RoboDK station: Pick and Place TT.rdk

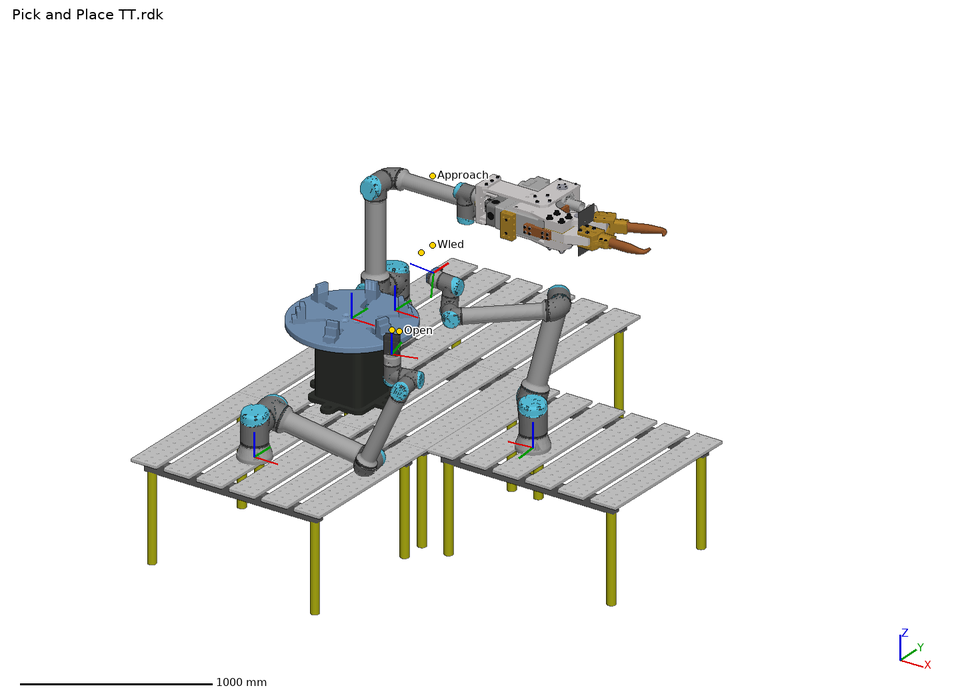
[picture v0: the station drawn from its stored meshes, robots at their saved joint values, targets as dots, program paths as lines]
Station Pick and Place (saved by RoboDK 5.6.0). Poses are relative to the parent item; angles as X-Y-Z fixed-axis rotations.
  - object Table at (1940, 2070, 0) mm, size 1193.8 x 965.2 x 609.6 mm, geometry from welding_table.sld
  - object Table at (740, 2070, 0) mm, size 1193.8 x 965.2 x 609.6 mm, geometry from welding_table.sld
  - object Table at (740, 3040, 0) mm, size 1193.8 x 965.2 x 609.6 mm, geometry from welding_table.sld
  - object Table at (740, 1100, 0) mm, size 1193.8 x 965.2 x 609.6 mm, geometry from welding_table.sld
  - frame UR10e Base at (660, 1000, 0) mm
    - robot UR10e: 6 axes, payload 10 kg, reach 1300 mm, repeatability 0.05 mm, weight 28.9 kg
        modified DH rows (alpha deg, a mm, theta deg, d mm): 0, 0, 0, 180.7; 90, 0, 180, 0; 0, 612.6, 0, 0; 0, 571.335, 0, 174.15; -90, 0, 0, 119.85; 90, 0, 180, 116.55
        joint limits [-360, -360, -360, -360, -360, -360] to [360, 360, 360, 360, 360, 360]; home [0, -90, -90, 0, 90, 0]; saved at [-169.455, 15.075, 278.893, 156.033, -90, 93.779]
      - frame Zimmer GEP2016IO-12-B-01 Gripper Base at (0, 0, 0) mm
        - robot Zimmer GEP2016IO-12-B-01 Gripper: 1 axes
            joint limits [0] to [40]; home [0]; saved at [0]
        - target Open (Cartesian target) at (40, 0, 140) mm; joints [0, -90, -90, 0, 90, 0] of UR10e
        - target Close (Cartesian target) at (0, 0, 140) mm; joints [0, -90, -90, 0, 90, 0] of UR10e
      - tool Tool 4, TCP at (0, 0, 140) mm
  - frame Welding at (260, 2840, 0) mm
    - robot UR10e-Welding (model UR10e): 6 axes, payload 10 kg, reach 1300 mm, repeatability 0.05 mm, weight 28.9 kg
        modified DH rows (alpha deg, a mm, theta deg, d mm): 0, 0, 0, 180.7; 90, 0, 180, 0; 0, 612.6, 0, 0; 0, 571.335, 0, 174.15; -90, 0, 0, 119.85; 90, 0, 180, 116.55
        joint limits [-360, -360, -360, -360, -360, -360] to [360, 360, 360, 360, 360, 360]; home [0, -90, -90, 0, 90, 0]; saved at [0, -90, -90, 0, 90, 0]
      - tool WeldGun3Dref, TCP at (0.14, 0, 525) mm, rotated rx 0 ry -90 rz 0 deg, size 252.3 x 125 x 530.5 mm
      - tool WeldGun, TCP at (0.27, 0, 1049.99) mm, rotated rx 0 ry -90 rz 0 deg
      - robot HMDTech_SpotWeld_Gun: 1 axes, payload 10 kg, repeatability 0.1 mm
          modified DH rows (alpha deg, a mm, theta deg, d mm): 0, 0, 0, 0
          base shift (0, 0, 600) mm, rotated rx 90 ry 0 rz 0 deg
          joint limits [-1] to [22.5]; home [0]; saved at [22.5]
      - tool Tool 4, TCP at (0, 0, 1050) mm
    - target Wled (Cartesian target) at (660, -600, 800) mm, rotated rx 0 ry 0 rz 14.32 deg; joints [100, 100, 100, 0, 0, 0, 10, 20, 30] of UR10e
    - target Approach (Cartesian target) at (660, -600, 1200) mm, rotated rx 0 ry 0 rz 14.32 deg; joints [100, 100, 100, 0, 0, 0, 10, 20, 30] of UR10e
    - target Wled (Cartesian target) at (660, -700, 800) mm, rotated rx 0 ry 0 rz 104.32 deg; joints [100, 100, 100, 0, 0, 0, 10, 20, 30] of UR10e
    - target Approach (Cartesian target) at (660, -600, 1200) mm, rotated rx 0 ry 0 rz 14.32 deg; joints [100, 100, 100, 0, 0, 0, 10, 20, 30] of UR10e
    - target Wled (Cartesian target) at (660, -700, 800) mm, rotated rx 0 ry 0 rz 90 deg; joints [100, 100, 100, 0, 0, 0, 10, 20, 30] of UR10e
    - target Approach (Cartesian target) at (660, -600, 1200) mm, rotated rx 0 ry 0 rz 14.32 deg; joints [100, 100, 100, 0, 0, 0, 10, 20, 30] of UR10e
  - frame TurnTable Base at (660, 1880, 450) mm
    - robot TurnTable: 1 axes
        modified DH rows (alpha deg, a mm, theta deg, d mm): 0, 0, 0, 0
        joint limits [-360] to [360]; home [0]; saved at [0]
    - frame staticRef at (0, 0, 0) mm
  - frame UR10e Base at (1780, 1920, 0) mm, rotated rx 0 ry 0 rz -175 deg
    - robot UR10e: 6 axes, payload 10 kg, reach 1300 mm, repeatability 0.05 mm, weight 28.9 kg
        modified DH rows (alpha deg, a mm, theta deg, d mm): 0, 0, 0, 180.7; 90, 0, 180, 0; 0, 612.6, 0, 0; 0, 571.335, 0, 174.15; -90, 0, 0, 119.85; 90, 0, 180, 116.55
        joint limits [-360, -360, -360, -360, -360, -360] to [360, 360, 360, 360, 360, 360]; home [0, -90, -90, 0, 90, 0]; saved at [32.677, -76.413, -106.374, 8.846, 54.41, -2.386]
      - frame Camera Ref Frame at (46.69, 0, 27.39) mm
        - object SICK VSPP-5F2113 Camera at (0, 0, 0) mm, size 116 x 53 x 38 mm, geometry from SICK-VSPP-5F2113-Camera.sld
